// Device/Application/Visu/Storage_Scheme_new
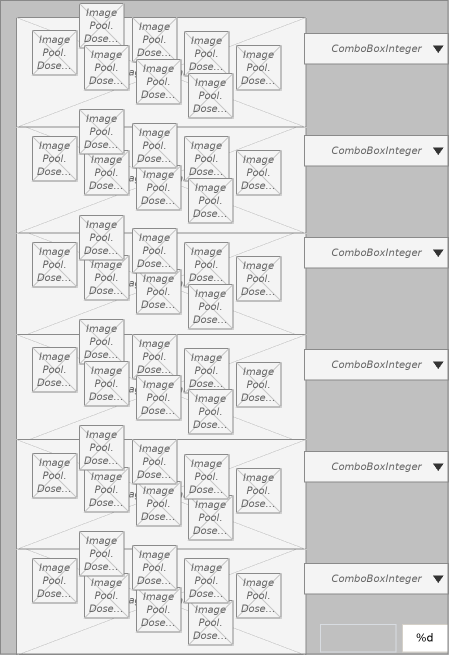
VISUALIZATION Storage_Scheme_new  // 449x655
    Image (16,228 290x110), image: ImagePool.Palette
    Image (184,242 45x45), invisible if: aStorePlace[3,2,0].aXVisability[2], image: ImagePool.Dose_silber
    Image (184,242 45x45), invisible if: aStorePlace[3,2,0].aXvisability[3], image: ImagePool.Dose_transparent
    Image (184,242 45x45), invisible if: aStorePlace[3,2,0].aXvisability[1], image: ImagePool.Dose_schwarz
    Image (184,242 45x45), invisible if: aStorePlace[3,2,0].aXvisability[0], image: ImagePool.Dose_rot
    Image (16,334 290x110), image: ImagePool.Palette
    Image (132,334 45x45), invisible if: aStorePlace[2,1,0].aXvisability[1], image: ImagePool.Dose_schwarz
    Image (132,334 45x45), invisible if: aStorePlace[2,1,0].aXvisability[2], image: ImagePool.Dose_silber
    Image (132,334 45x45), invisible if: aStorePlace[2,1,0].aXvisability[3], image: ImagePool.Dose_transparent
    Image (132,334 45x45), invisible if: aStorePlace[2,1,0].aXvisability[0], image: ImagePool.Dose_rot
    Image (16,545 290x110), image: ImagePool.Palette
    Image (16,439 290x110), image: ImagePool.Palette
    Image (16,123 290x110), image: ImagePool.Palette
    Image (16,17 290x110), image: ImagePool.Palette
    Image (236,45 45x45), invisible if: aStorePlace[5,3,0].aXvisability[2], image: ImagePool.Dose_silber
    Image (236,45 45x45), invisible if: aStorePlace[5,3,0].aXvisability[3], image: ImagePool.Dose_transparent
    Image (236,45 45x45), invisible if: aStorePlace[5,3,0].aXvisability[1], image: ImagePool.Dose_schwarz
    Image (236,45 45x45), invisible if: aStorePlace[5,3,0].aXvisability[0], image: ImagePool.Dose_rot
    Image (184,31 45x45), invisible if: aStorePlace[5,2,0].aXvisability[2], image: ImagePool.Dose_silber
    Image (184,31 45x45), invisible if: aStorePlace[5,2,0].aXvisability[3], image: ImagePool.Dose_transparent
    Image (184,31 45x45), invisible if: aStorePlace[5,2,0].aXvisability[1], image: ImagePool.Dose_schwarz
    Image (184,31 45x45), invisible if: aStorePlace[5,2,0].aXvisability[0], image: ImagePool.Dose_rot
    Image (132,17 45x45), invisible if: aStorePlace[5,1,0].aXvisability[2], image: ImagePool.Dose_silber
    Image (132,17 45x45), invisible if: aStorePlace[5,1,0].aXvisability[3], image: ImagePool.Dose_transparent
    Image (132,17 45x45), invisible if: aStorePlace[5,1,0].aXvisability[1], image: ImagePool.Dose_schwarz
    Image (132,17 45x45), invisible if: aStorePlace[5,1,0].aXvisability[0], image: ImagePool.Dose_rot
    Image (79,3 45x45), invisible if: aStorePlace[5,0,0].aXvisability[2], image: ImagePool.Dose_silber
    Image (79,3 45x45), invisible if: aStorePlace[5,0,0].aXvisability[3], image: ImagePool.Dose_transparent
    Image (79,3 45x45), invisible if: aStorePlace[5,0,0].aXvisability[1], image: ImagePool.Dose_schwarz
    Image (79,3 45x45), invisible if: aStorePlace[5,0,0].aXvisability[0], image: ImagePool.Dose_rot
    Image (32,30 45x45), invisible if: aStorePlace[5,0,1].aXvisability[2], image: ImagePool.Dose_silber
    Image (32,30 45x45), invisible if: aStorePlace[5,0,1].aXvisability[3], image: ImagePool.Dose_transparent
    Image (32,30 45x45), invisible if: aStorePlace[5,0,1].aXvisability[1], image: ImagePool.Dose_schwarz
    Image (32,30 45x45), invisible if: aStorePlace[5,0,1].aXvisability[0], image: ImagePool.Dose_rot
    Image (84,45 45x45), invisible if: aStorePlace[5,1,1].aXvisability[2], image: ImagePool.Dose_silber
    Image (84,45 45x45), invisible if: aStorePlace[5,1,1].aXvisability[3], image: ImagePool.Dose_transparent
    Image (84,45 45x45), invisible if: aStorePlace[5,1,1].aXvisability[1], image: ImagePool.Dose_schwarz
    Image (84,45 45x45), invisible if: aStorePlace[5,1,1].aXvisability[0], image: ImagePool.Dose_rot
    Image (136,59 45x45), invisible if: aStorePlace[5,2,1].aXvisability[2], image: ImagePool.Dose_silber
    Image (136,59 45x45), invisible if: aStorePlace[5,2,1].aXvisability[3], image: ImagePool.Dose_transparent
    Image (136,59 45x45), invisible if: aStorePlace[5,2,1].aXvisability[1], image: ImagePool.Dose_schwarz
    Image (136,59 45x45), invisible if: aStorePlace[5,2,1].aXvisability[0], image: ImagePool.Dose_rot
    Image (188,73 45x45), invisible if: aStorePlace[5,3,1].aXvisability[2], image: ImagePool.Dose_silber
    Image (188,73 45x45), invisible if: aStorePlace[5,3,1].aXvisability[3], image: ImagePool.Dose_transparent
    Image (188,73 45x45), invisible if: aStorePlace[5,3,1].aXvisability[1], image: ImagePool.Dose_schwarz
    Image (188,73 45x45), invisible if: aStorePlace[5,3,1].aXvisability[0], image: ImagePool.Dose_rot
    Image (136,165 45x45), invisible if: aStorePlace[4,2,1].aXvisability[2], image: ImagePool.Dose_silber
    Image (136,165 45x45), invisible if: aStorePlace[4,2,1].aXvisability[3], image: ImagePool.Dose_transparent
    Image (136,165 45x45), invisible if: aStorePlace[4,2,1].aXvisability[1], image: ImagePool.Dose_schwarz
    Image (136,165 45x45), invisible if: aStorePlace[4,2,1].aXvisability[0], image: ImagePool.Dose_rot
    Image (84,150 45x45), invisible if: aStorePlace[4,1,1].aXvisability[2], image: ImagePool.Dose_silber
    Image (84,150 45x45), invisible if: aStorePlace[4,1,1].aXvisability[3], image: ImagePool.Dose_transparent
    Image (84,150 45x45), invisible if: aStorePlace[4,1,1].aXvisability[1], image: ImagePool.Dose_schwarz
    Image (84,150 45x45), invisible if: aStorePlace[4,1,1].aXvisability[0], image: ImagePool.Dose_rot
    Image (32,136 45x45), invisible if: aStorePlace[4,0,1].aXvisability[2], image: ImagePool.Dose_silber
    Image (32,136 45x45), invisible if: aStorePlace[4,0,1].aXvisability[3], image: ImagePool.Dose_transparent
    Image (32,136 45x45), invisible if: aStorePlace[4,0,1].aXvisability[1], image: ImagePool.Dose_schwarz
    Image (32,136 45x45), invisible if: aStorePlace[4,0,1].aXvisability[0], image: ImagePool.Dose_rot
    Image (79,109 45x45), invisible if: aStorePlace[4,0,0].aXvisability[2], image: ImagePool.Dose_silber
    Image (79,109 45x45), invisible if: aStorePlace[4,0,0].aXvisability[3], image: ImagePool.Dose_transparent
    Image (79,109 45x45), invisible if: aStorePlace[4,0,0].aXvisability[1], image: ImagePool.Dose_schwarz
    Image (79,109 45x45), invisible if: aStorePlace[4,0,0].aXvisability[0], image: ImagePool.Dose_rot
    Image (132,123 45x45), invisible if: aStorePlace[4,1,0].aXvisability[2], image: ImagePool.Dose_silber
    Image (132,123 45x45), invisible if: aStorePlace[4,1,0].aXvisability[3], image: ImagePool.Dose_transparent
    Image (132,123 45x45), invisible if: aStorePlace[4,1,0].aXvisability[1], image: ImagePool.Dose_schwarz
    Image (132,123 45x45), invisible if: aStorePlace[4,1,0].aXvisability[0], image: ImagePool.Dose_rot
    Image (184,136 45x45), invisible if: aStorePlace[4,2,0].aXvisability[2], image: ImagePool.Dose_silber
    Image (184,136 45x45), invisible if: aStorePlace[4,2,0].aXvisability[3], image: ImagePool.Dose_transparent
    Image (184,136 45x45), invisible if: aStorePlace[4,2,0].aXvisability[1], image: ImagePool.Dose_schwarz
    Image (184,136 45x45), invisible if: aStorePlace[4,2,0].aXvisability[0], image: ImagePool.Dose_rot
    Image (236,150 45x45), invisible if: aStorePlace[4,3,0].aXvisability[2], image: ImagePool.Dose_silber
    Image (236,150 45x45), invisible if: aStorePlace[4,3,0].aXvisability[3], image: ImagePool.Dose_transparent
    Image (236,150 45x45), invisible if: aStorePlace[4,3,0].aXvisability[1], image: ImagePool.Dose_schwarz
    Image (236,150 45x45), invisible if: aStorePlace[4,3,0].aXvisability[0], image: ImagePool.Dose_rot
    Image (188,178 45x45), invisible if: aStorePlace[4,3,1].aXvisability[2], image: ImagePool.Dose_silber
    Image (188,178 45x45), invisible if: aStorePlace[4,3,1].aXvisability[3], image: ImagePool.Dose_transparent
    Image (188,178 45x45), invisible if: aStorePlace[4,3,1].aXvisability[1], image: ImagePool.Dose_schwarz
    Image (188,178 45x45), invisible if: aStorePlace[4,3,1].aXvisability[0], image: ImagePool.Dose_rot
    Image (84,255 45x45), invisible if: aStorePlace[3,2,1].aXvisability[2], image: ImagePool.Dose_silber
    Image (84,255 45x45), invisible if: aStorePlace[3,2,1].aXvisability[3], image: ImagePool.Dose_transparent
    Image (84,255 45x45), invisible if: aStorePlace[3,2,1].aXvisability[1], image: ImagePool.Dose_schwarz
    Image (84,255 45x45), invisible if: aStorePlace[3,2,1].aXvisability[0], image: ImagePool.Dose_rot
    Image (136,269 45x45), invisible if: aStorePlace[3,2,1].aXvisability[2], image: ImagePool.Dose_silber
    Image (136,269 45x45), invisible if: aStorePlace[3,2,1].aXvisability[3], image: ImagePool.Dose_transparent
    Image (136,269 45x45), invisible if: aStorePlace[3,2,1].aXvisability[1], image: ImagePool.Dose_schwarz
    Image (136,269 45x45), invisible if: aStorePlace[3,2,1].aXvisability[0], image: ImagePool.Dose_rot
    Image (188,284 45x45), invisible if: aStorePlace[3,3,1].aXvisability[2], image: ImagePool.Dose_silber
    Image (188,284 45x45), invisible if: aStorePlace[3,3,1].aXvisability[3], image: ImagePool.Dose_transparent
    Image (188,284 45x45), invisible if: aStorePlace[3,3,1].aXvisability[1], image: ImagePool.Dose_schwarz
    Image (188,284 45x45), invisible if: aStorePlace[3,3,1].aXvisability[0], image: ImagePool.Dose_rot
    Image (236,256 45x45), invisible if: aStorePlace[3,3,0].aXvisability[2], image: ImagePool.Dose_silber
    Image (236,256 45x45), invisible if: aStorePlace[3,3,0].aXvisability[3], image: ImagePool.Dose_transparent
    Image (236,256 45x45), invisible if: aStorePlace[3,3,0].aXvisability[1], image: ImagePool.Dose_schwarz
    Image (236,256 45x45), invisible if: aStorePlace[3,3,0].aXvisability[0], image: ImagePool.Dose_rot
    Image (132,228 45x45), invisible if: aStorePlace[3,1,0].aXvisability[2], image: ImagePool.Dose_silber
    Image (132,228 45x45), invisible if: aStorePlace[3,1,0].aXvisability[3], image: ImagePool.Dose_transparent
    Image (132,228 45x45), invisible if: aStorePlace[3,1,0].aXvisability[1], image: ImagePool.Dose_schwarz
    Image (132,228 45x45), invisible if: aStorePlace[3,1,0].aXvisability[0], image: ImagePool.Dose_rot
    Image (32,242 45x45), invisible if: aStorePlace[3,0,1].aXvisability[2], image: ImagePool.Dose_silber
    Image (32,242 45x45), invisible if: aStorePlace[3,0,1].aXvisability[3], image: ImagePool.Dose_transparent
    Image (32,242 45x45), invisible if: aStorePlace[3,0,1].aXvisability[1], image: ImagePool.Dose_schwarz
    Image (32,242 45x45), invisible if: aStorePlace[3,0,1].aXvisability[0], image: ImagePool.Dose_rot
    Image (79,215 45x45), invisible if: aStorePlace[3,0,0].aXvisability[2], image: ImagePool.Dose_silber
    Image (79,215 45x45), invisible if: aStorePlace[3,0,0].aXvisability[3], image: ImagePool.Dose_transparent
    Image (79,215 45x45), invisible if: aStorePlace[3,0,0].aXvisability[1], image: ImagePool.Dose_schwarz
    Image (79,215 45x45), invisible if: aStorePlace[3,0,0].aXvisability[0], image: ImagePool.Dose_rot
    Image (79,319 45x45), invisible if: aStorePlace[2,0,0].aXvisability[2], image: ImagePool.Dose_silber
    Image (79,319 45x45), invisible if: aStorePlace[2,0,0].aXvisability[3], image: ImagePool.Dose_transparent
    Image (79,319 45x45), invisible if: aStorePlace[2,0,0].aXvisability[1], image: ImagePool.Dose_schwarz
    Image (79,319 45x45), invisible if: aStorePlace[2,0,0].aXvisability[0], image: ImagePool.Dose_rot
    Image (79,319 45x45), invisible if: aStorePlace[2,0,0].aXvisability[2], image: ImagePool.Dose_silber
    Image (79,319 45x45), invisible if: aStorePlace[2,0,0].aXvisability[3], image: ImagePool.Dose_transparent
    Image (79,319 45x45), invisible if: aStorePlace[2,0,0].aXvisability[1], image: ImagePool.Dose_schwarz
    Image (79,319 45x45), invisible if: aStorePlace[2,0,0].aXvisability[0], image: ImagePool.Dose_rot
    Image (184,348 45x45), invisible if: aStorePlace[2,2,0].aXvisability[2], image: ImagePool.Dose_silber
    Image (184,348 45x45), invisible if: aStorePlace[2,2,0].aXvisability[3], image: ImagePool.Dose_transparent
    Image (184,348 45x45), invisible if: aStorePlace[2,2,0].aXvisability[1], image: ImagePool.Dose_schwarz
    Image (184,348 45x45), invisible if: aStorePlace[2,2,0].aXvisability[0], image: ImagePool.Dose_rot
    Image (236,362 45x45), invisible if: aStorePlace[2,3,0].aXvisability[2], image: ImagePool.Dose_silber
    Image (236,362 45x45), invisible if: aStorePlace[2,3,0].aXvisability[3], image: ImagePool.Dose_transparent
    Image (236,362 45x45), invisible if: aStorePlace[2,3,0].aXvisability[1], image: ImagePool.Dose_schwarz
    Image (236,362 45x45), invisible if: aStorePlace[2,3,0].aXvisability[0], image: ImagePool.Dose_rot
    Image (188,389 45x45), invisible if: aStorePlace[2,3,1].aXvisability[2], image: ImagePool.Dose_silber
    Image (188,389 45x45), invisible if: aStorePlace[2,3,1].aXvisability[3], image: ImagePool.Dose_transparent
    Image (188,389 45x45), invisible if: aStorePlace[2,3,1].aXvisability[1], image: ImagePool.Dose_schwarz
    Image (188,389 45x45), invisible if: aStorePlace[2,3,1].aXvisability[0], image: ImagePool.Dose_rot
    Image (136,375 45x45), invisible if: aStorePlace[2,2,1].aXvisability[2], image: ImagePool.Dose_silber
    Image (136,375 45x45), invisible if: aStorePlace[2,2,1].aXvisability[3], image: ImagePool.Dose_transparent
    Image (136,375 45x45), invisible if: aStorePlace[2,2,1].aXvisability[1], image: ImagePool.Dose_schwarz
    Image (136,375 45x45), invisible if: aStorePlace[2,2,1].aXvisability[0], image: ImagePool.Dose_rot
    Image (84,361 45x45), invisible if: aStorePlace[2,1,1].aXvisability[2], image: ImagePool.Dose_silber
    Image (84,361 45x45), invisible if: aStorePlace[2,1,1].aXvisability[3], image: ImagePool.Dose_transparent
    Image (84,361 45x45), invisible if: aStorePlace[2,1,1].aXvisability[1], image: ImagePool.Dose_schwarz
    Image (84,361 45x45), invisible if: aStorePlace[2,1,1].aXvisability[0], image: ImagePool.Dose_rot
    Image (32,347 45x45), invisible if: aStorePlace[2,0,1].aXvisability[2], image: ImagePool.Dose_silber
    Image (32,347 45x45), invisible if: aStorePlace[2,0,1].aXvisability[3], image: ImagePool.Dose_transparent
    Image (32,347 45x45), invisible if: aStorePlace[2,0,1].aXvisability[1], image: ImagePool.Dose_schwarz
    Image (32,347 45x45), invisible if: aStorePlace[2,0,1].aXvisability[0], image: ImagePool.Dose_rot
    Image (32,453 45x45), invisible if: aStorePlace[1,0,1].aXvisability[2], image: ImagePool.Dose_silber
    Image (32,453 45x45), invisible if: aStorePlace[1,0,1].aXvisability[3], image: ImagePool.Dose_transparent
    Image (32,453 45x45), invisible if: aStorePlace[1,0,1].aXvisability[1], image: ImagePool.Dose_schwarz
    Image (32,453 45x45), invisible if: aStorePlace[1,0,1].aXvisability[0], image: ImagePool.Dose_rot
    Image (84,467 45x45), invisible if: aStorePlace[1,1,1].aXvisability[2], image: ImagePool.Dose_silber
    Image (84,467 45x45), invisible if: aStorePlace[1,1,1].aXvisability[3], image: ImagePool.Dose_transparent
    Image (84,467 45x45), invisible if: aStorePlace[1,1,1].aXvisability[1], image: ImagePool.Dose_schwarz
    Image (84,467 45x45), invisible if: aStorePlace[1,1,1].aXvisability[0], image: ImagePool.Dose_rot
    Image (136,481 45x45), invisible if: aStorePlace[1,2,1].aXvisability[2], image: ImagePool.Dose_silber
    Image (136,481 45x45), invisible if: aStorePlace[1,2,1].aXvisability[3], image: ImagePool.Dose_transparent
    Image (136,481 45x45), invisible if: aStorePlace[1,2,1].aXvisability[1], image: ImagePool.Dose_schwarz
    Image (136,481 45x45), invisible if: aStorePlace[1,2,1].aXvisability[0], image: ImagePool.Dose_rot
    Image (188,495 45x45), invisible if: aStorePlace[1,3,1].aXvisability[2], image: ImagePool.Dose_silber
    Image (188,495 45x45), invisible if: aStorePlace[1,3,1].aXvisability[3], image: ImagePool.Dose_transparent
    Image (188,495 45x45), invisible if: aStorePlace[1,3,1].aXvisability[1], image: ImagePool.Dose_schwarz
    Image (188,495 45x45), invisible if: aStorePlace[1,3,1].aXvisability[0], image: ImagePool.Dose_rot
    Image (236,468 45x45), invisible if: aStorePlace[1,3,0].aXvisability[2], image: ImagePool.Dose_silber
    Image (236,468 45x45), invisible if: aStorePlace[1,3,0].aXvisability[3], image: ImagePool.Dose_transparent
    Image (236,468 45x45), invisible if: aStorePlace[1,3,0].aXvisability[1], image: ImagePool.Dose_schwarz
    Image (236,468 45x45), invisible if: aStorePlace[1,3,0].aXvisability[0], image: ImagePool.Dose_rot
    Image (184,454 45x45), invisible if: aStorePlace[1,2,0].aXvisability[2], image: ImagePool.Dose_silber
    Image (184,454 45x45), invisible if: aStorePlace[1,2,0].aXvisability[3], image: ImagePool.Dose_transparent
    Image (184,454 45x45), invisible if: aStorePlace[1,2,0].aXvisability[1], image: ImagePool.Dose_schwarz
    Image (184,454 45x45), invisible if: aStorePlace[1,2,0].aXvisability[0], image: ImagePool.Dose_rot
    Image (132,439 45x45), invisible if: aStorePlace[1,1,0].aXvisability[2], image: ImagePool.Dose_silber
    Image (132,439 45x45), invisible if: aStorePlace[1,1,0].aXvisability[0], image: ImagePool.Dose_transparent
    Image (79,425 45x45), invisible if: aStorePlace[1,0,0].aXvisability[2], image: ImagePool.Dose_silber
    Image (79,425 45x45), invisible if: aStorePlace[1,0,0].aXvisability[3], image: ImagePool.Dose_transparent
    Image (79,425 45x45), invisible if: aStorePlace[1,0,0].aXvisability[1], image: ImagePool.Dose_schwarz
    Image (79,425 45x45), invisible if: aStorePlace[1,0,0].aXvisability[0], image: ImagePool.Dose_rot
    Image (188,600 45x45), invisible if: aStorePlace[0,3,1].aXvisability[2], image: ImagePool.Dose_silber
    Image (188,600 45x45), invisible if: aStorePlace[0,3,1].aXvisability[3], image: ImagePool.Dose_transparent
    Image (188,600 45x45), invisible if: aStorePlace[0,3,1].aXvisability[1], image: ImagePool.Dose_schwarz
    Image (132,439 45x45), invisible if: aStorePlace[1,1,0].aXVisability[1], image: ImagePool.Dose_schwarz
    Image (188,600 45x45), invisible if: aStorePlace[0,3,1].aXvisability[0], image: ImagePool.Dose_rot
    Image (132,439 45x45), invisible if: aStorePlace[1,1,0].aXvisability[0], image: ImagePool.Dose_rot
    Image (136,587 45x45), invisible if: aStorePlace[0,2,1].aXvisability[2], image: ImagePool.Dose_silber
    Image (136,587 45x45), invisible if: aStorePlace[0,2,1].aXvisability[3], image: ImagePool.Dose_transparent
    Image (136,587 45x45), invisible if: aStorePlace[0,2,1].aXvisability[1], image: ImagePool.Dose_schwarz
    Image (136,587 45x45), invisible if: aStorePlace[0,2,1].aXvisability[0], image: ImagePool.Dose_rot
    Image (84,573 45x45), invisible if: aStorePlace[0,1,1].aXvisability[2], image: ImagePool.Dose_silber
    Image (84,573 45x45), invisible if: aStorePlace[0,1,1].aXvisability[3], image: ImagePool.Dose_transparent
    Image (84,573 45x45), invisible if: aStorePlace[0,1,1].aXvisability[1], image: ImagePool.Dose_schwarz
    Image (84,573 45x45), invisible if: aStorePlace[0,1,1].aXvisability[0], image: ImagePool.Dose_rot
    Image (32,558 45x45), invisible if: aStorePlace[0,0,1].aXvisability[2], image: ImagePool.Dose_silber
    Image (32,558 45x45), invisible if: aStorePlace[0,0,1].aXvisability[3], image: ImagePool.Dose_transparent
    Image (32,558 45x45), invisible if: aStorePlace[0,0,1].aXvisability[1], image: ImagePool.Dose_schwarz
    Image (32,558 45x45), invisible if: aStorePlace[0,0,1].aXvisability[0], image: ImagePool.Dose_rot
    Image (79,531 45x45), invisible if: aStorePlace[0,0,0].aXvisability[2], image: ImagePool.Dose_silber
    Image (79,531 45x45), invisible if: aStorePlace[0,0,0].aXvisability[3], image: ImagePool.Dose_transparent
    Image (79,531 45x45), invisible if: aStorePlace[0,0,0].aXvisability[1], image: ImagePool.Dose_schwarz
    Image (79,531 45x45), invisible if: aStorePlace[0,0,0].aXVisability[0], image: ImagePool.Dose_rot
    Image (132,545 45x45), invisible if: aStorePlace[0,1,0].aXVisability[2], image: ImagePool.Dose_silber
    Image (132,545 45x45), invisible if: aStorePlace[0,1,0].aXVisability[3], image: ImagePool.Dose_transparent
    Image (132,545 45x45), invisible if: aStorePlace[0,1,0].aXVisability[1], image: ImagePool.Dose_schwarz
    Image (132,545 45x45), invisible if: aStorePlace[0, 1, 0].aXVisability[0], image: ImagePool.Dose_rot
    Image (184,558 45x45), invisible if: aStorePlace[0,2,0].aXVisability[2], image: ImagePool.Dose_silber
    Image (184,558 45x45), invisible if: aStorePlace[0,2,0].aXVisability[3], image: ImagePool.Dose_transparent
    Image (184,558 45x45), invisible if: aStorePlace[0,2,0].aXVisability[1], image: ImagePool.Dose_schwarz
    Image (184,558 45x45), invisible if: aStorePlace[0,2,0].aXVisability[0], image: ImagePool.Dose_rot
    Image (184,558 45x45), invisible if: aStorePlace[0,2,0].aXVisability[2], image: ImagePool.Dose_silber
    Image (184,558 45x45), invisible if: aStorePlace[0,2,0].aXVisability[3], image: ImagePool.Dose_transparent
    Image (184,558 45x45), invisible if: aStorePlace[0,2,0].aXVisability[1], image: ImagePool.Dose_schwarz
    Image (184,558 45x45), invisible if: aStorePlace[0,2,0].aXVisability[0], image: ImagePool.Dose_rot
    Image (236,573 45x45), invisible if: aStorePlace[0,3,0].aXVisability[2], image: ImagePool.Dose_silber
    Image (236,573 45x45), invisible if: aStorePlace[0,3,0].aXVisability[3], image: ImagePool.Dose_transparent
    Image (236,573 45x45), invisible if: aStorePlace[0,3,0].aXVisability[1], image: ImagePool.Dose_schwarz
    Image (236,573 45x45), invisible if: aStorePlace[0,3,0].aXVisability[0], image: ImagePool.Dose_rot
    ComboBoxInteger (304,33 145x31), variable: aUIColorChoose[5], text list: 'ARR_COLORCHOOSE'
        p1601986498: 'ImagePool'
    ComboBoxInteger (304,135 145x31), variable: aUIColorChoose[4], text list: 'ARR_COLORCHOOSE'
        p1601986498: 'ImagePool'
    ComboBoxInteger (304,237 145x31), variable: aUIColorChoose[3], text list: 'ARR_COLORCHOOSE'
        p1601986498: 'ImagePool'
    ComboBoxInteger (304,349 145x31), variable: aUIColorChoose[2], text list: 'ARR_COLORCHOOSE'
        p1601986498: 'ImagePool'
    ComboBoxInteger (304,451 145x31), variable: aUIColorChoose[1], text list: 'ARR_COLORCHOOSE'
        p1601986498: 'ImagePool'
    ComboBoxInteger (304,563 145x31), variable: aUIColorChoose[0], text list: 'ARR_COLORCHOOSE'
        p1601986498: 'ImagePool'
    Rectangle (320,624 76x28), text list: 'Glob_TextList', text index: '129'
    Textfield (402,624 46x28), "%d", text variable: bBitCount
END_VISUALIZATION

// Device/Application/Visu/Optionen
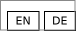
VISUALIZATION Optionen  // 76x31
    Rectangle (7,11 32x20), "EN", text list: 'Glob_TextList', text index: '3'
        OnMouseDown:  ChangeLanguage=Englisch
    Rectangle (44,11 32x20), "DE", text list: 'Glob_TextList', text index: '3'
        OnMouseDown:  ChangeLanguage=Deutsch
END_VISUALIZATION

// Device/Application/Visu/StorageVisu
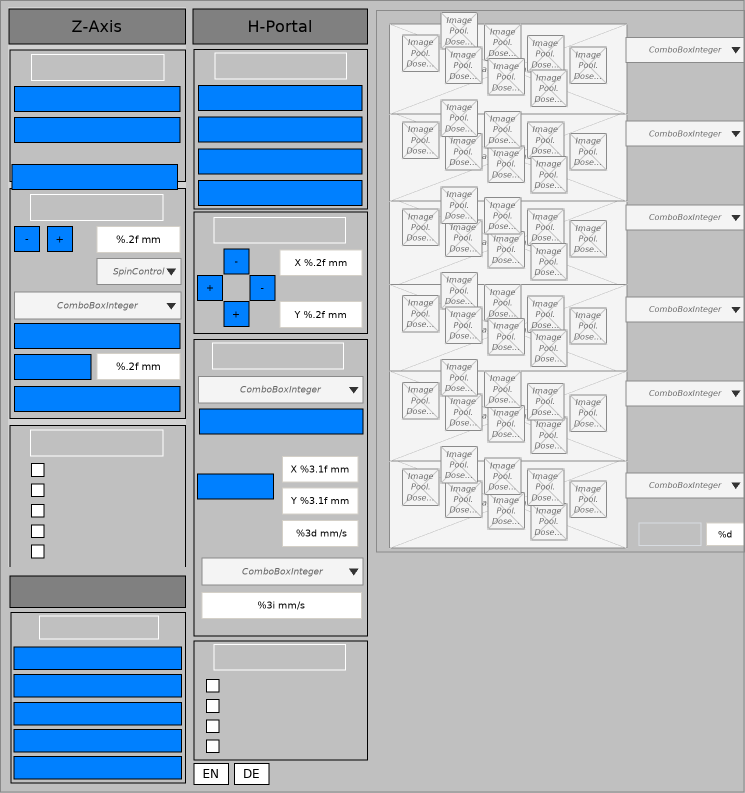
VISUALIZATION StorageVisu  // 745x793
    Frame (8,7 254x561)
        shows Z_Axis()
    Frame (376,10 369x542)
        shows Storage_Scheme_new()
    Frame (192,8 219x752)
        shows H_Portal()
    Frame (186,751 83x42)
        shows Optionen()
    Frame (1,567 189x218)
        shows generalControls()
END_VISUALIZATION

// Device/Application/Visu/H_Portal
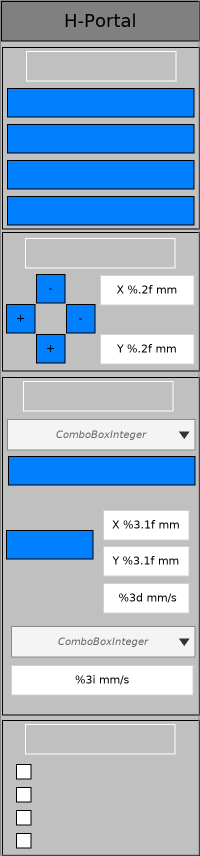
VISUALIZATION H_Portal  // 200x856
    Rectangle (2,232 198x139)
    Rectangle (2,720 198x136)
    Rectangle (6,304 29x29), "+", input disabled if: xEnAuto OR NOT xStatusGlobalReference
        tap xManuVisuJogPosY
    Rectangle (66,304 29x29), "-", input disabled if: xEnAuto OR NOT xStatusGlobalReference
        tap xManuVisuJogNegY
    Rectangle (1,1 199x40), "H-Portal"
    Textfield (100,275 94x30), "X %.2f mm", text variable: rPOSX_Ausgabe
    Rectangle (25,238 150x30), text list: 'Glob_TextList', text index: '105'
    Rectangle (25,724 150x30), text list: 'Glob_TextList', text index: '106'
    Rectangle (2,47 198x182)
    Rectangle (7,88 187x29), input disabled if: xEXCM_HOMED, text list: 'Glob_TextList', text index: '109'
        tap xHomeExcm
    Rectangle (26,51 150x30), text list: 'Glob_TextList', text index: '110'
    Rectangle (7,160 187x29), text list: 'Glob_TextList', text index: '107'
        tap xEXCM_Res_Fault p1329445385=TRUE
    Rectangle (7,124 187x29), text list: 'Glob_TextList', text index: '108'
        toggle xEXCM_En_Drive
    Textfield (100,334 94x30), "Y %.2f mm", text variable: rPOSY_Ausgabe
    Rectangle (36,274 29x29), "-", input disabled if: xEnAuto OR NOT xStatusGlobalReference
        tap xManuVisuJogNegX
    Rectangle (36,334 29x29), "+", input disabled if: xEnAuto OR NOT xStatusGlobalReference
        tap xManuVisuJogPosX
    Rectangle (16,764 15x15), colour toggle: xEXCM_STATUS_DriveEnabled
    Rectangle (16,810 15x15), colour toggle: xEXCM_STATUS_RefPointReached
    Rectangle (16,833 15x15), colour toggle: xEXCM_STATUS_Fault
    Rectangle (16,787 15x15), colour toggle: xEXCM_STATUS_VoltagePresent
    Rectangle (40,782 122x20), text list: 'Glob_TextList', text index: '103'
    Rectangle (40,205 122x20), text list: 'Glob_TextList', text index: '101'
    Rectangle (40,828 122x20), text list: 'Glob_TextList', text index: '104'
    Rectangle (40,759 122x20), text list: 'Glob_TextList', text index: '102'
    Rectangle (2,377 198x338)
    Rectangle (23,381 150x30), text list: 'Glob_TextList', text index: '112'
    Rectangle (6,530 87x29), input disabled if: xEnAuto, text list: 'Glob_TextList', text index: '112'
        tap xTeachXY
    ComboBoxInteger (7,419 188x31), variable: usiVisabilityXYOptions, text list: 'ARR_XYPOS'
    Rectangle (8,456 187x29), input disabled if: xEnAuto, text list: 'Glob_TextList', text index: '117'
        tap xDriveManualXYPos
    ComboBoxInteger (11,626 184x31), variable: usiVisabilitySpeedOptions, text list: 'ARR_XYPOS'
    Textfield (11,665 182x30), "%3i mm/s", text variable: uiLayOnSpeed, invisible if: aXVisabilitySpeedOptions[3]
        OnMouseClick: write the text variable via Default, min 1, max 30
    Textfield (11,665 182x30), "%3i mm/s", text variable: uiGrabSpeed, invisible if: aXVisabilitySpeedOptions[2]
        OnMouseClick: write the text variable via Default, min 1, max 50
    Textfield (11,665 182x30), "%3i mm/s", text variable: uiDriveSpeed, invisible if: aXVisabilitySpeedOptions[1]
        OnMouseClick: write the text variable via Default, min 1, max 200
    Textfield (103,510 86x30), "X %3.1f mm", text variable: rXPositionGrab, invisible if: aXVisabilityXYPositions[1], input disabled if: xEnAuto
        OnMouseClick: write the text variable via Default, min 1, max 599
    Textfield (103,546 86x30), "Y %3.1f mm", text variable: rYPositionGrab, invisible if: aXVisabilityXYPositions[1], input disabled if: xEnAuto
        OnMouseClick: write the text variable via Default, min 0, max 209
    Textfield (103,510 86x30), "X %3.1f mm", text variable: rXPositionIdle, invisible if: aXVisabilityXYPositions[2], input disabled if: xEnAuto
        OnMouseClick: write the text variable via Default, min 1, max 599
    Textfield (103,546 86x30), "Y %3.1f mm", text variable: rYPositionIdle, invisible if: aXVisabilityXYPositions[2], input disabled if: xEnAuto
        OnMouseClick: write the text variable via Default, min 0, max 209
    Textfield (103,510 86x30), "X %3.1f mm", text variable: rXPositionWorkPiece1, invisible if: aXVisabilityXYPositions[4], input disabled if: xEnAuto
        OnMouseClick: write the text variable via Default, min 1, max 599
    Textfield (103,546 86x30), "Y %3.1f mm", text variable: rYPositionWorkPiece1, invisible if: aXVisabilityXYPositions[4], input disabled if: xEnAuto
        OnMouseClick: write the text variable via Default, min 0, max 209
    Textfield (103,510 86x30), "X %3.1f mm", text variable: rXPositionTransfer, invisible if: aXVisabilityXYPositions[3], input disabled if: xEnAuto
        OnMouseClick: write the text variable via Default, min 1, max 599
    Textfield (103,546 86x30), "Y %3.1f mm", text variable: rYPositionTransfer, invisible if: aXVisabilityXYPositions[3], input disabled if: xEnAuto
        OnMouseClick: write the text variable via Default, min 0, max 209
    Rectangle (8,586 94x22), text list: 'Glob_TextList', text index: '118'
    Textfield (103,583 86x30), "%3d mm/s", text variable: uiVisuVelocity, input disabled if: xEnAuto
        OnMouseClick: write the text variable via Default, min 0, max 209
    Rectangle (7,196 187x29), text list: 'Glob_TextList', text index: '122'
        tap xEXCM_Stop_Drive p1329445385=TRUE
    Rectangle (40,810 122x20), text list: 'Glob_TextList', text index: '101'
END_VISUALIZATION

// Device/Application/Visu/Z_Axis
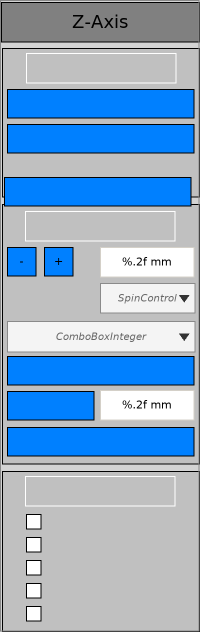
VISUALIZATION Z_Axis  // 200x632
    Rectangle (2,204 198x260)
    Rectangle (2,471 198x161)
    Rectangle (44,247 29x29), "+", input disabled if: xEnAuto OR NOT xStatusGlobalReference
        tap xTapForward
    Rectangle (7,247 29x29), "-", input disabled if: xEnAuto OR NOT xStatusGlobalReference
        tap xTapBackward
    Rectangle (1,2 199x40), "Z-Axis"
    Textfield (100,247 94x30), "%.2f mm", text variable: cmmoSTAxis.lrCurrentPos
        OnMouseClick: write the text variable via Default, min 0, max 250
    Rectangle (26,514 15x15), colour toggle: CMMO_POWER_1.xEnabled
    Rectangle (25,211 150x30), text list: 'Glob_TextList', text index: '105'
    Rectangle (25,476 150x30), text list: 'Glob_TextList', text index: '106'
    Rectangle (2,48 198x149)
    Rectangle (7,89 187x29), input disabled if: xEnAuto OR xStatusGlobalReference, text list: 'Glob_TextList', text index: '109'
        tap xHomeZAxis
    Rectangle (26,53 150x30), text list: 'Glob_TextList', text index: '110'
    Rectangle (7,124 187x29), text list: 'Glob_TextList', text index: '107'
        tap CMMO_RESET_1.xExecute
    Rectangle (26,560 15x15), colour toggle: CMMO_SW.xReferenced
    Rectangle (26,583 15x15), colour toggle: CMMO_DRIVER_1.xError
    Rectangle (26,606 15x15), colour toggle: CMMO_DRIVER_1.xIsConnected
    Rectangle (26,537 15x15), colour toggle: CMMO_POWER_1.xEnabled
    Rectangle (49,509 122x20), text list: 'Glob_TextList', text index: '102'
    Rectangle (49,532 122x20), text list: 'Glob_TextList', text index: '103'
    Rectangle (49,555 122x20), text list: 'Glob_TextList', text index: '101'
    Rectangle (49,578 122x20), text list: 'Glob_TextList', text index: '104'
    Rectangle (49,601 122x20), text list: 'Glob_TextList', text index: '114'
    Textfield (100,390 94x30), "%.2f mm", text variable: lrZPositionGrab, invisible if: aXVisabilityZPositions[1]
    Textfield (100,390 94x30), "%.2f mm", text variable: lrZPositionWorkPieceFront, invisible if: aXVisabilityZPositions[2]
    Textfield (100,390 94x30), "%.2f mm", text variable: lrZPositionWorkPieceRear, invisible if: aXVisabilityZPositions[3]
    Rectangle (7,391 87x29), input disabled if: xEnAuto OR NOT xStatusGlobalReference, text list: 'Glob_TextList', text index: '112'
        tap xTeach
    Rectangle (11,324 85x20), text list: 'Glob_TextList', text index: '113'
    Rectangle (4,177 187x29), input disabled if: CMMO_DRIVER_1.xIsConnected, text list: 'Glob_TextList', text index: '111'
        toggle xConnectCMMO
    ComboBoxInteger (7,321 188x31), variable: usiVisabilityZOptions, text list: 'ARR_ZPOS'
    SpinControl (100,283 95x30), variable: lrStepSize
        p1653691745: 0.1
        OnMouseClick: write the text variable via Default, min 0.1, max 10
    Rectangle (5,288 91x20), text list: 'Glob_TextList', text index: '115'
    Rectangle (7,356 187x29), text list: 'Glob_TextList', text index: '116'
        OnMouseClick:  ToggleVariable=xReadPositionsOnce
    Rectangle (7,427 187x29), input disabled if: xEnAuto OR NOT xStatusGlobalReference, text list: 'Glob_TextList', text index: '117'
        OnMouseClick: execute { xDriveZManual := TRUE; }
END_VISUALIZATION

// Device/Application/Visu/generalControls
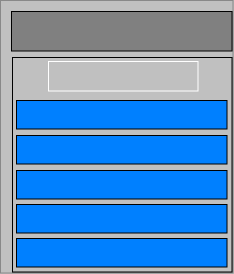
VISUALIZATION generalControls  // 234x274
    Rectangle (11,11 221x40), text list: 'Glob_TextList', text index: '119'
    Rectangle (12,57 220x215)
    Rectangle (16,100 211x29), input disabled if: xStatusGlobalReference, text list: 'Glob_TextList', text index: '120'
        OnMouseClick:  ToggleVariable=xGlobalReference
    Rectangle (48,61 150x30), text list: 'Glob_TextList', text index: '110'
    Rectangle (16,170 211x29), text list: 'Glob_TextList', text index: '100'
        OnMouseClick:  ToggleVariable=xGlobalReset
    Rectangle (16,135 211x29), input disabled if: xEnAuto, text list: 'Glob_TextList', text index: '121'
        OnMouseClick:  ToggleVariable=qxGrab
    Rectangle (16,204 211x29), text list: 'Glob_TextList', text index: '127'
        OnMouseClick:  ToggleVariable=xClearStore
    Rectangle (16,238 211x29), input disabled if: NOT xStatusGlobalReference, text list: 'Glob_TextList', text index: '128'
        OnMouseClick:  ToggleVariable=xEnAuto
END_VISUALIZATION

(* text list Glob_TextList (id | default | Englisch | Deutsch)
  1 | Deutsch | Englisch | Deutsch
  101 | xReferenziert | xReferenced | xReferenziert
  102 | xFreigabe | xEnabled | xFreigabe
  103 | x24V Versorgung | x24V Power | x24V Versorgung
  104 | xFehler | xError | xFehler
  105 | Manuelles tippen | Manual Jogging | Manuelles tippen
  106 | Status | Status | Status
  107 | Fehler quittieren | Reset Error | Fehler quittieren
  108 | Aktivieren | Enable | Aktivieren
  109 | Referenzieren | Home | Referenzieren
  110 | Manuelle Steuerung | Manual Control | Manuelle Steuerung
  111 | Verbinden | Connect | Verbinden
  112 | Pos. Speichern | Teach Pos. | Pos. Speichern
  113 | Position | Position	 | Position
  114 | xVerbunden | xConnected | xVerbunden
  115 | Schrittweite | Stepsize | Schrittweite
  116 | Positionen lesen | Read Positions | Positionen lesen
  117 | Position fahren | Drive position | Position fahren
  118 | Man. Geschw. | Man. Velocity | Man. Geschw.
  119 | Allg. Kontrolle | General Controls | Allg. Kontrolle
  120 | Kompl. Referenzieren | Global reference | Kompl. Referenzieren
  121 | Greifen | Grab | Greifen
  122 | Stoppen | Stop | Stoppen
  123 | rot | red | rot
  124 | schwarz | black | schwarz
  125 | silber | silver | silber
  126 | transparent | transparent | transparent
  127 | Lager leeren | Clear Store | Lager leeren
  128 | Auto/Manuell | Auto/Manual | Auto/Manuell
  100 | Kompl. Reset | Global Reset | Kompl. Reset
  129 | BitSelection | Bit selection | Bit Auswahl
   |  |  |  *)

(* text list ARR_ZPOS (id | default | Englisch | Deutsch)
  1 | Abholposition | Grab position | Abholposition
  2 | Pos. WS vorne | Pos. WS front | Pos. WS vorne
  3 | Pos. WS hinten | Pos. WS rear | Pos. WS hinten
   |  |  |  *)

(* text list ARR_XYPOS (id | default | Englisch | Deutsch)
  1 | Abholposition | Grab Position | Abholposition
  2 | Warteposition | Idle Position | Warteposition
  3 | Ablageposition | Transfer Position | Ablageposition
  4 | Position Werkst.1 | Position Workp. | Position Werkst.
   |  |  |  *)

(* text list ARR_SPEED (id | default | Englisch | Deutsch)
  1 | Geschw. Fahren | Vel. drive | Geschw. Fahren
  2 | Geschw. Greifen | Vel. grab | Geschw. Greifen
  3 | Geschw. WS Greifen | Vel. grab Workpiece | Geschw. WS greifen
   |  |  |  *)

(* text list ARR_COLORCHOOSE (id | default | Englisch | Deutsch)
  0 | rot | red | rot
  1 | schwarz | black | schwarz
  2 | silber | silver | silber
  3 | transparent | transparent | transparent
   |  |  |  *)
